FUNCTION F_ToArrInterlocks : ARRAY[1..8] OF BOOL
VAR_INPUT
	In1		:BOOL;
	In2		:BOOL;
	In3		:BOOL;
	In4		:BOOL;
	In5		:BOOL;
	In6		:BOOL;
	In7		:BOOL;
	In8		:BOOL;
END_VAR
VAR
END_VAR

F_ToArrInterlocks[1] := In1;
F_ToArrInterlocks[2] := In2;
F_ToArrInterlocks[3] := In3;
F_ToArrInterlocks[4] := In4;
F_ToArrInterlocks[5] := In5;
F_ToArrInterlocks[6] := In6;
F_ToArrInterlocks[7] := In7;
F_ToArrInterlocks[8] := In8;

END_FUNCTION

(* stored: Version 1.1.0.1, ProductVersion 3.1.4024.12
   POU F_ToArrInterlocks: Id {1dbebe28-7f60-416e-aaf9-2a2b24858c28}, SpecialFunc None *)
